# EPICS autosave request: iocBoot/ioc-test/autosave/auto_settings.req
file "sample_settings.req", P=IOC:autosave:, N=sample_positioner
IOC:ACF:Test
IOC:ACF:LI:OPSTATE
IOC:ACF:LI:lev1permit
IOC:STREAM:checksum
file configMenu_settings.req P=$(P),CONFIG=scan1
